TYPE E_EPT :
(
	// Unknown, Alarm, Paused, Aborting, Claibration, Manual
	eBlocked :=0,
	// Idle
	eIdle,
	// Initialize, SettingUp, Ready, Executing, Checking
	eBusy 
);
END_TYPE

(* stored: Version 1.1.0.1, ProductVersion 3.1.4022.12
   DUT E_EPT: Id {b182f51e-d1ce-408a-90e1-2ef0dc5a69eb} *)
